{attribute 'TcGenerated'}
{attribute 'no-analysis'}
{attribute 'linkalways'}
// This function has been automatically generated from the project information.
VAR_GLOBAL CONSTANT
	{attribute 'const_non_replaced'}
	stLibVersion_tcl_StringUtils : ST_LibVersion := (iMajor := 1, iMinor := 1, iBuild := 7, iRevision := 0, nFlags := 0, sVersion := '1.1.7.0');
END_VAR

(* stored: Version 1.1.0.1, ProductVersion 3.1.4024.15
   GVL Global_Version: Id {6efc34ee-d4b3-4312-ada8-56d0e461983a} *)
